Omron CX-Programmer project NewProject (CX-Programmer 9.75)

# PLC NewPLC1: CP1E E20

## Global symbols (name address type ; comment)
0.08 BOOL  ; sensor sorting optic
0.11 BOOL  ; Auto man
0.07 BOOL  ; sensor benda sorting
0.09 BOOL  ; sensor sorting induktif
0.10 BOOL  ; sensor seluncuran
0.12 BOOL  ; pb start
W50.00 BOOL  ; workpiece silver
W50.01 BOOL  ; workpiece merah
W50.02 BOOL  ; workpiece hitam

## Program NewProgram1 (cyclic task 0)

### Section Section1

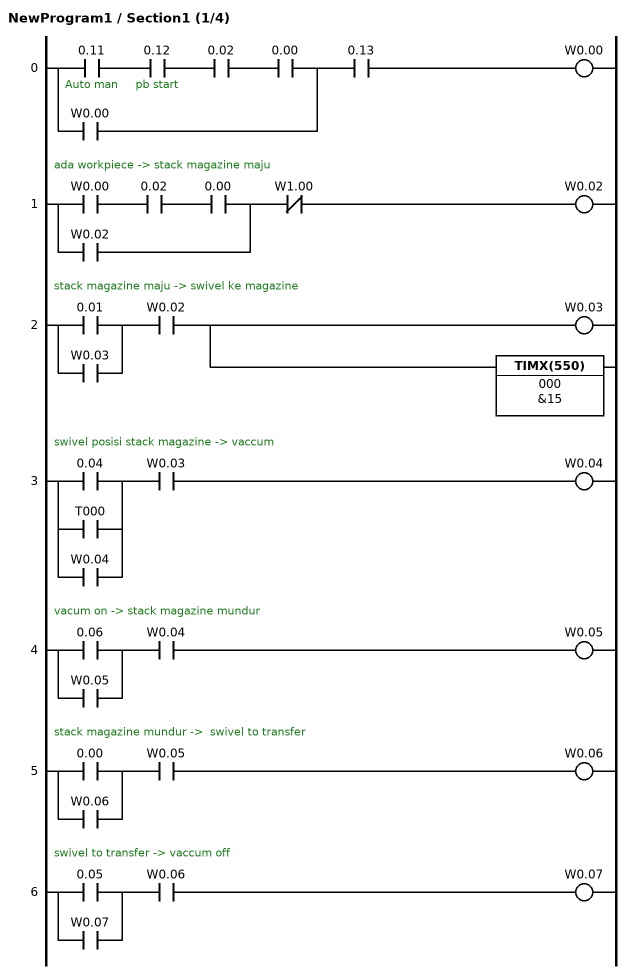
; rung 0
LD 0.11  ; Auto man
AND 0.12  ; pb start
AND 0.02
AND 0.00
OR W0.00
AND 0.13
OUT W0.00
; rung 1: ada workpiece -> stack magazine maju
LD W0.00
AND 0.02
AND 0.00
OR W0.02
ANDNOT W1.00
OUT W0.02
; rung 2: stack magazine maju -> swivel ke magazine
LD 0.01
OR W0.03
AND W0.02
OUT W0.03
TIMX(550) 000 &15
; rung 3: swivel posisi stack magazine -> vaccum
LD 0.04
OR T000
OR W0.04
AND W0.03
OUT W0.04
; rung 4: vacum on -> stack magazine mundur
LD 0.06
OR W0.05
AND W0.04
OUT W0.05
; rung 5: stack magazine mundur ->  swivel to transfer
LD 0.00
OR W0.06
AND W0.05
OUT W0.06
; rung 6: swivel to transfer -> vaccum off
LD 0.05
OR W0.07
AND W0.06
OUT W0.07

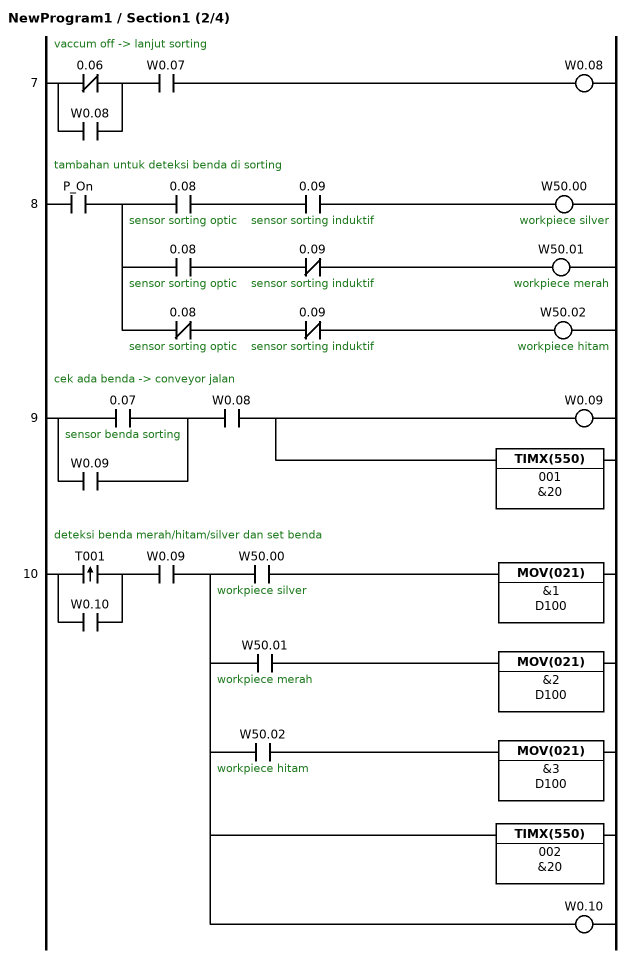
; rung 7: vaccum off -> lanjut sorting
LDNOT 0.06
OR W0.08
AND W0.07
OUT W0.08
; rung 8: tambahan untuk deteksi benda di sorting
LD P_On
OUT TR0
AND 0.08  ; sensor sorting optic
AND 0.09  ; sensor sorting induktif
OUT W50.00  ; workpiece silver
LD TR0
AND 0.08  ; sensor sorting optic
ANDNOT 0.09  ; sensor sorting induktif
OUT W50.01  ; workpiece merah
LD TR0
ANDNOT 0.08  ; sensor sorting optic
ANDNOT 0.09  ; sensor sorting induktif
OUT W50.02  ; workpiece hitam
; rung 9: cek ada benda -> conveyor jalan
LD 0.07  ; sensor benda sorting
OR W0.09
AND W0.08
OUT W0.09
TIMX(550) 001 &20
; rung 10: deteksi benda merah/hitam/silver dan set benda
@LD T001
OR W0.10
AND W0.09
OUT TR0
AND W50.00  ; workpiece silver
MOV(021) &1 D100
LD TR0
AND W50.01  ; workpiece merah
MOV(021) &2 D100
LD TR0
AND W50.02  ; workpiece hitam
MOV(021) &3 D100
LD TR0
TIMX(550) 002 &20
OUT W0.10

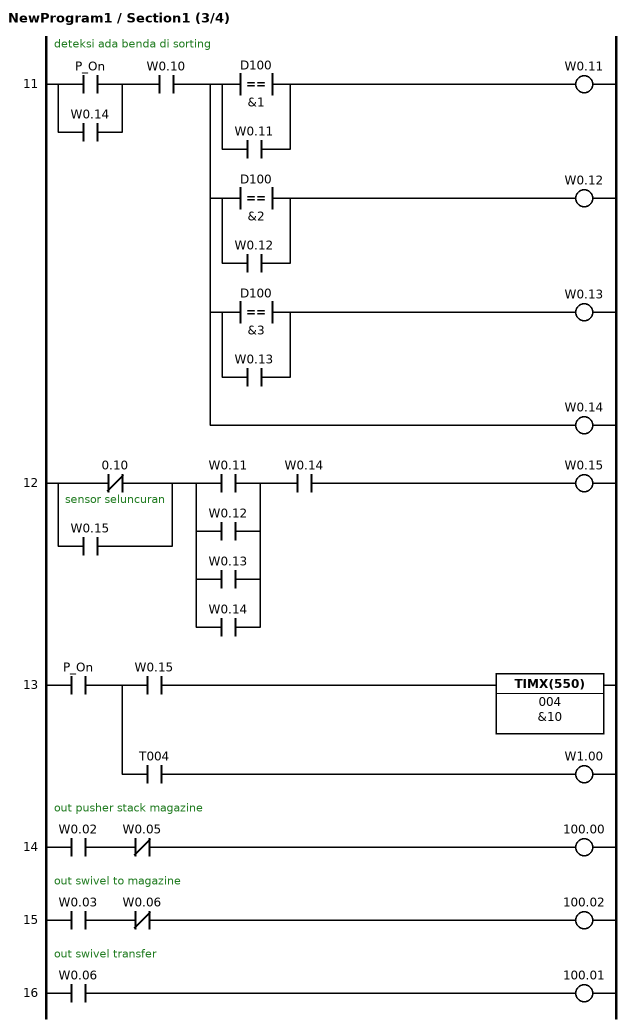
; rung 11: deteksi ada benda di sorting
LD P_On
OR W0.14
AND W0.10
OUT TR0
LD=(300) D100 &1
OR W0.11
ANDLD
OUT W0.11
LD TR0
LD=(300) D100 &2
OR W0.12
ANDLD
OUT W0.12
LD TR0
LD=(300) D100 &3
OR W0.13
ANDLD
OUT W0.13
LD TR0
OUT W0.14
; rung 12
LDNOT 0.10  ; sensor seluncuran
OR W0.15
LD W0.11
OR W0.12
OR W0.13
OR W0.14
ANDLD
AND W0.14
OUT W0.15
; rung 13
LD P_On
OUT TR0
AND W0.15
TIMX(550) 004 &10
LD TR0
AND T004
OUT W1.00
; rung 14: out pusher stack magazine
LD W0.02
ANDNOT W0.05
OUT 100.00
; rung 15: out swivel to magazine
LD W0.03
ANDNOT W0.06
OUT 100.02
; rung 16: out swivel transfer
LD W0.06
OUT 100.01

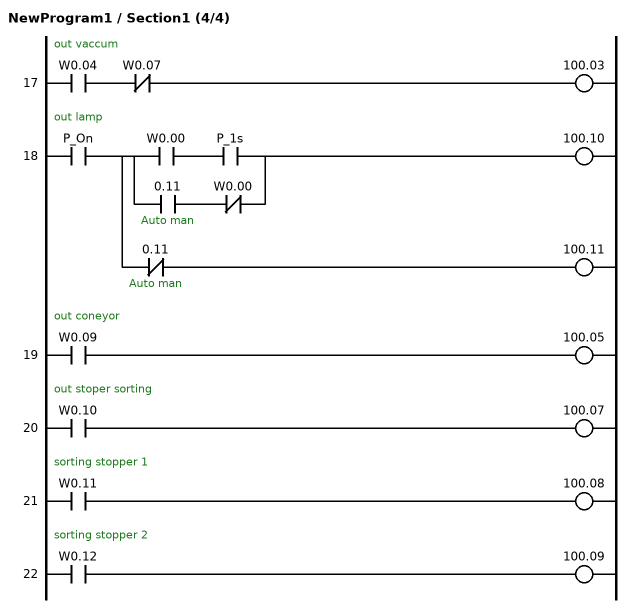
; rung 17: out vaccum
LD W0.04
ANDNOT W0.07
OUT 100.03
; rung 18: out lamp
LD P_On
OUT TR0
LD W0.00
AND P_1s
LD 0.11  ; Auto man
ANDNOT W0.00
ORLD
ANDLD
OUT 100.10
LD TR0
ANDNOT 0.11  ; Auto man
OUT 100.11
; rung 19: out coneyor
LD W0.09
OUT 100.05
; rung 20: out stoper sorting
LD W0.10
OUT 100.07
; rung 21: sorting stopper 1
LD W0.11
OUT 100.08
; rung 22: sorting stopper 2
LD W0.12
OUT 100.09

### Section END
; rung 0
END(001)